// TwinCAT 3 PLC project Lynus_Test
// ProgramVersion: 3.1.4023.0
// libraries:
//   EfficientIO Communicator, * (EfficientIO)
//   EfficientIO ModbusTCP, * (EfficientIO)
//   Lynus Standards, * (Lynus AG)
//   Tc2_ModbusSrv, * (Beckhoff Automation GmbH)
//   Tc2_Standard, * (Beckhoff Automation GmbH)
//   Tc2_System, * (Beckhoff Automation GmbH)
//   Tc2_Utilities, * (Beckhoff Automation GmbH)
//   Tc3_Module, * (Beckhoff Automation GmbH)
//   Lynus Energy Basic,1.0.0.2,Lynus AG
// project tree:
//   DUTs/ st_P_Connect_to_Lynus.TcDUT
//   GVLs/ GVL.TcGVL, p_Datenschnittstelle_L.TcPOU
//   Lynus/ EfficientIO_Read_Wirte.TcPOU, MqttCommunicator.TcPOU, PrgEMS.TcPOU, PrgModbus.TcPOU, p_call_fast_task.TcPOU, p_slow_task.TcPOU
//   / EfficientIO_Communication.TcTTO, PlcTask1.TcTTO
// (motion and I/O tree: see PLC project p_connect)
// real-time tasks:
//   TASK PlcTask: cycle T#10ms, priority 20, ADS port 350
//   TASK EfficientIO_Communication: cycle T#5ms, priority 15, ADS port 351
//   TASK PlcTask1: cycle T#10ms, priority 21, ADS port 353
// variable links:
//   Lynus_Test/Lynus_Test Instance <-> P_Connect/P_Connect Instance
//     PlcTask1 Inputs/GVL.lynus_in <-> PlcTask Outputs/GVL_EfficientIO.lynus_out
//     PlcTask1 Outputs/GVL.lynus_out <-> PlcTask Inputs/GVL_EfficientIO.lynus_in

CONFIGURATION Lynus_Test
    RESOURCE PLC ON TwinCAT3
        TASK EfficientIO_Communication(INTERVAL := T#5ms, PRIORITY := 15);
        TASK PlcTask1(INTERVAL := T#10ms, PRIORITY := 21);
        PROGRAM p_call_fast_task WITH EfficientIO_Communication : p_call_fast_task;
        PROGRAM p_slow_task WITH PlcTask1 : p_slow_task;
    END_RESOURCE
END_CONFIGURATION

// ---- DUTs/st_P_Connect_to_Lynus.TcDUT
TYPE st_P_Connect_to_Lynus :
STRUCT
	Wert_1	:REAL;	
	Wert_2	:REAL;	
	Wert_3	:REAL;	
	Wert_4	:REAL;	
	Wert_5	:REAL;	
	Wert_6	:REAL;	
	Wert_7	:BOOL;	
	Wert_8	:REAL;	
	Wert_9	:REAL;	
	Wert_10	:REAL;
	Wert_11	:REAL;	
	Wert_12	:REAL;	
	Wert_13	:REAL;	
	Wert_14	:REAL;	
	Wert_15	:REAL;	
	Wert_16	:REAL;	
	Wert_17	:REAL;	
	Wert_18	:REAL;	
	Wert_19	:REAL;	
	Wert_20	:REAL;
	Wert_21	:REAL;	
	Wert_22	:REAL;	
	Wert_23	:REAL;	
	Wert_24	:REAL;	
	Wert_25	:REAL;	
	Wert_26	:REAL;	
	Wert_27	:REAL;	
	Wert_28	:REAL;	
	Wert_29	:REAL;	
	Wert_30	:REAL;
	Wert_31	:REAL;
	Wert_32	:REAL;
	Wert_33	:REAL;
	Wert_34	:REAL;
	Wert_35	:REAL;
	Wert_36	:REAL;
	Wert_37	:REAL;
	Wert_38	:REAL;
	Wert_39	:REAL;
	Wert_40	:REAL;
	Wert_41	:BOOL;
	Wert_42	:BOOL;
	Wert_43	:BOOL;
	Wert_44	:BOOL;
	Wert_45	:BOOL;
	Wert_46	:BOOL;
	Wert_47	:BOOL;
	Wert_48	:BOOL;
	Wert_49	:BOOL;
	Wert_50	:BOOL;
	Wert_51	:BOOL;
	Wert_52	:BOOL;
END_STRUCT
END_TYPE

// ---- GVLs/GVL.TcGVL
{attribute 'qualified_only'}
VAR_GLOBAL
	lynus_in   				AT %I* 	: st_P_Connect_to_Lynus;
	lynus_out   			AT %Q* 	: st_P_Connect_to_Lynus;
	
	NULL						:REAL;//{#lynus.ag#()}
	
	(*KNX*)
	TEMP_INNEN_1					:REAL;//{#lynus.ag#()}
	RH_INNEN_1						:REAL;//{#lynus.ag#()}
	TEMP_INNEN_2					:REAL;//{#lynus.ag#()}
	RH_INNEN_2						:REAL;//{#lynus.ag#()}
	TEMP_AUSSEN						:REAL;//{#lynus.ag#()}
	RH_AUSSEN						:REAL;//{#lynus.ag#()}
	AKTIVITAET						:BOOL;//{#lynus.ag#()}
	
	(*M-Bus variablen für Lynus*)
	ELEKTRO_1_Zaehler		:REAL;//{#lynus.ag#()}
	ELEKTRO_1_Leistung		:REAL;//{#lynus.ag#()}
	ELEKTRO_2_Zaehler		:REAL;//{#lynus.ag#()}
	ELEKTRO_2_Leistung		:REAL;//{#lynus.ag#()}
	ELEKTRO_3_Zaehler		:REAL;//{#lynus.ag#()}
	ELEKTRO_3_Leistung		:REAL;//{#lynus.ag#()}
	ELEKTRO_4_Zaehler		:REAL;//{#lynus.ag#()}
	ELEKTRO_4_Leistung		:REAL;//{#lynus.ag#()}
	ELEKTRO_5_Zaehler		:REAL;//{#lynus.ag#()}
	ELEKTRO_5_Leistung		:REAL;//{#lynus.ag#()}
	HEIZEN					:REAL;//{#lynus.ag#()}
	HEIZEN_E_Lesitung		:REAL;//{#lynus.ag#()}
	
	(*IMPULSZÄHLER*)
	Wasseruhr_1				:REAL;//{#lynus.ag#()}
	Wasseruhr_2				:REAL;//{#lynus.ag#()}

	(*PT1000 Temp.*)
	TEMP_HKLS_1				:REAL;//{#lynus.ag#()}
	TEMP_HKLS_2				:REAL;//{#lynus.ag#()}
	TEMP_HKLS_3				:REAL;//{#lynus.ag#()}
	TEMP_HKLS_4				:REAL;//{#lynus.ag#()}
	TEMP_HKLS_5				:REAL;//{#lynus.ag#()}
	TEMP_HKLS_6				:REAL;//{#lynus.ag#()}
	TEMP_HKLS_7				:REAL;//{#lynus.ag#()}
	TEMP_HKLS_8				:REAL;//{#lynus.ag#()}
	
	(*Zentalfunktionen*)
	VERSCHATTUNG_auf		:BOOL;//{#lynus.ag#()}
	VERSCHATTUNG_ab			:BOOL;//{#lynus.ag#()}
	ZENTRAL_LICHT_ein_EG	:BOOL;//{#lynus.ag#()}
	ZENTRAL_LICHT_aus_EG	:BOOL;//{#lynus.ag#()}
	ZENTRAL_LICHT_ein_OG	:BOOL;//{#lynus.ag#()}
	ZENTRAL_LICHT_aus_OG	:BOOL;//{#lynus.ag#()}
	B3_ZENTRAL_LICHT_ein	:BOOL;//{#lynus.ag#()}
	B3_ZENTRAL_LICHT_aus	:BOOL;//{#lynus.ag#()}
	B3_SCHATTUNG_auf_EG		:BOOL;//{#lynus.ag#()}
	B3_SCHATTUNG_ab_EG		:BOOL;//{#lynus.ag#()}
	B3_SCHATTUNG_auf_OG		:BOOL;//{#lynus.ag#()}
	B3_SCHATTUNG_ab_OG		:BOOL;//{#lynus.ag#()}
	
	Wert_30					:REAL;//{#lynus.ag#()}
	Wert_31					:REAL;//{#lynus.ag#()}
	Wert_32					:REAL;//{#lynus.ag#()}
	Wert_33					:REAL;//{#lynus.ag#()}
	dummy_					:BOOL;//{#lynus.ag#()}
END_VAR

// ---- Lynus/p_call_fast_task.TcPOU
PROGRAM p_call_fast_task
VAR
	EfficientIO: INT;
END_VAR

(* Es wird standartmäßig M-Bus verwendet, bei IMMODO wurden Mod-Bus zähler verbaut *)
//Communication_KL6781();
(*MAIN_Zaehlerbaustein()*);

(*FB's von Lynus die den FastTask bennötigen*)
EfficientIO_Read_Wirte();

END_PROGRAM

// ---- Lynus/EfficientIO_Read_Wirte.TcPOU
PROGRAM EfficientIO_Read_Wirte
VAR
	fbVar				: FB_VarInfo;
	fbRW				: FB_ReadWrite;
END_VAR

(*Der FB_VarInfo sammelt die Informationen über alle kommentierten Variablen in der SPS.*)
fbVar(
	bReadInfo:= , 
	eTMCFile:= eSelectTMCFile.eDontUseTMCFile, 
	eSavePositionTMCFile:= eSavePositionOnPLC.ePostionC, 
	udiCounterFoundVariables=> , 
	bError=> , 
	bBusy=> , 
	byProgress=> , 
	udiErrorCodeOut=> , 
	eErrorVarInfo_Out=> , 
	sVarWithError=> );

(*Der FB_ReadWrite dient nach dem Scannen der Symbole dem Lesen und Schreiben der Werte.
Die gelesenen Werte werden in Richtung Cloud geschickt und die schreibenden, kommend von
der Cloud, werden auf den Wert der SPS geschrieben.*)
fbrw();

END_PROGRAM

// ---- Lynus/p_slow_task.TcPOU
PROGRAM p_slow_task
VAR
END_VAR

(*Programmaufrufte im slow Task (10ms)*)
//Call Slow Tasks for Lynus 	
MqttCommunicator();
p_Datenschnittstelle_L();


//Stefan Lackner 14.02.2023
PrgModbus();		// Modbus TCP functions
PrgEMS();			// EMS Fucntion

END_PROGRAM

// ---- Lynus/MqttCommunicator.TcPOU
PROGRAM MqttCommunicator
VAR
	fbCom			: FB_MqttCommunicator_V5;
END_VAR

(*notdonepoint Bitte UserName und UserPassword eintragen, dies bekommt man direkt von der LynusWebsite*)
fbCom(
	bConnect:= TRUE, 
	strAuthKey:= 'ENE87365342998', 
	sUserName:='7ad7b8b6-0630-4d31-a3b5-e626a3dca2b4', 
	sUserPassword:='b0a3873e-12bb-4efd-a1d1-df77771e0e45', 
	eSavePositionCertificate:= eSavePositionOnPLC.ePostionC, 
	bConnected=> , 
	bError=> , 
	hrErrorCode=> , 
	eConnectionState=> , 
	eErrorMessage_Out=> );

(*fbCom(
	bConnect:= TRUE, 
	sUserName:= '0d553fc2-e7f3-4571-9008-fb5428f4c828',
	sUserPassword:= '8604f195-2f00-444b-ac81-e02a496b91e8', 
	eSavePositionCertificate:= eSavePositionOnPLC.ePostionC, 
	bConnected=> , 
	bError=> , 
	hrErrorCode=> , 
	eConnectionState=> , 
	eErrorMessage_Out=> );
	*)

END_PROGRAM

// ---- GVLs/p_Datenschnittstelle_L.TcPOU
PROGRAM p_Datenschnittstelle_L
VAR
END_VAR

GVL.NULL				:=0.0;
GVL.TEMP_INNEN_1		:= GVL.lynus_in.Wert_1;	
GVL.RH_INNEN_1			:= GVL.lynus_in.Wert_2;
GVL.TEMP_INNEN_2		:= GVL.lynus_in.Wert_3;
GVL.RH_INNEN_2			:= GVL.lynus_in.Wert_4;
GVL.TEMP_AUSSEN			:= GVL.lynus_in.Wert_5;
GVL.RH_AUSSEN			:= GVL.lynus_in.Wert_6;
GVL.AKTIVITAET			:= GVL.lynus_in.Wert_7;
GVL.ELEKTRO_1_Zaehler	:= GVL.lynus_in.Wert_8;
GVL.ELEKTRO_1_Leistung	:= GVL.lynus_in.Wert_9;
GVL.ELEKTRO_2_Zaehler	:= GVL.lynus_in.Wert_10;
GVL.ELEKTRO_2_Leistung	:= GVL.lynus_in.Wert_11;
GVL.ELEKTRO_3_Zaehler	:= GVL.lynus_in.Wert_12;
GVL.ELEKTRO_3_Leistung	:= GVL.lynus_in.Wert_13;
GVL.ELEKTRO_4_Zaehler	:= GVL.lynus_in.Wert_14;
GVL.ELEKTRO_4_Leistung	:= GVL.lynus_in.Wert_15;
GVL.ELEKTRO_5_Zaehler	:= GVL.lynus_in.Wert_16;
GVL.ELEKTRO_5_Leistung	:= GVL.lynus_in.Wert_17;
GVL.HEIZEN				:= GVL.lynus_in.Wert_18;
GVL.HEIZEN_E_Lesitung	:= GVL.lynus_in.Wert_19;
GVL.Wasseruhr_1			:= GVL.lynus_in.Wert_20;
GVL.Wasseruhr_2			:= GVL.lynus_in.Wert_21;
GVL.TEMP_HKLS_1			:= GVL.lynus_in.Wert_22;
GVL.TEMP_HKLS_2			:= GVL.lynus_in.Wert_23;
GVL.TEMP_HKLS_3			:= GVL.lynus_in.Wert_24;
GVL.TEMP_HKLS_4			:= GVL.lynus_in.Wert_25;
GVL.TEMP_HKLS_5			:= GVL.lynus_in.Wert_26;
GVL.TEMP_HKLS_6			:= GVL.lynus_in.Wert_27;
GVL.TEMP_HKLS_7			:= GVL.lynus_in.Wert_28;
GVL.TEMP_HKLS_8			:= GVL.lynus_in.Wert_29;

GVL.Wert_30				:= GVL.lynus_in.Wert_30;
GVL.Wert_31				:= GVL.lynus_in.Wert_31; //BA3 WP Leistung
GVL.Wert_32				:= GVL.lynus_in.Wert_32; //BA3 WP Energie Wärme
GVL.Wert_33				:= GVL.lynus_in.Wert_33; //BA3 WP Energie Kälte

GVL.lynus_out.Wert_41	:= GVL.VERSCHATTUNG_auf;
GVL.lynus_out.Wert_42	:= GVL.VERSCHATTUNG_ab;
GVL.lynus_out.Wert_43	:= GVL.ZENTRAL_LICHT_ein_EG;
GVL.lynus_out.Wert_44	:= GVL.ZENTRAL_LICHT_aus_EG;
GVL.lynus_out.Wert_45	:= GVL.ZENTRAL_LICHT_ein_OG;
GVL.lynus_out.Wert_46	:= GVL.ZENTRAL_LICHT_aus_OG;
GVL.lynus_out.Wert_47	:= GVL.B3_ZENTRAL_LICHT_ein;
GVL.lynus_out.Wert_48	:= GVL.B3_ZENTRAL_LICHT_aus;
GVL.lynus_out.Wert_49	:= GVL.B3_SCHATTUNG_auf_EG;
GVL.lynus_out.Wert_50	:= GVL.B3_SCHATTUNG_ab_EG;
GVL.lynus_out.Wert_51	:= GVL.B3_SCHATTUNG_auf_OG;
GVL.lynus_out.Wert_52	:= GVL.B3_SCHATTUNG_ab_OG;

END_PROGRAM

// ---- Lynus/PrgModbus.TcPOU
PROGRAM PrgModbus
VAR
	FB_KEBA_CS1				:FB_ECS_KEBA_P30;
	FB_Schneider_EVLink_1	:FB_Schneider_EVlinkWallbox;
	FB_Schneider_EVLink_2	:FB_Schneider_EVlinkWallbox;
	FB_Schneider_EVLink_3	:FB_Schneider_EVlinkWallbox;
	FB_Schneider_EVLink_4	:FB_Schneider_EVlinkWallbox;
	FB_Schneider_EVLink_5	:FB_Schneider_EVlinkWallbox;
	FB_Schneider_EVLink_6	:FB_Schneider_EVlinkWallbox;
	FB_Schneider_EVLink_7	:FB_Schneider_EVlinkWallbox;
	FB_Schneider_EVLink_8	:FB_Schneider_EVlinkWallbox;
	FB_Schneider_EVLink_9	:FB_Schneider_EVlinkWallbox;
	FB_Schneider_EVLink_10	:FB_Schneider_EVlinkWallbox;
	FB_Schneider_EVLink_11	:FB_Schneider_EVlinkWallbox;
	FB_Schneider_EVLink_12	:FB_Schneider_EVlinkWallbox;
	FB_Schneider_EVLink_13	:FB_Schneider_EVlinkWallbox;
	FB_Schneider_EVLink_14	:FB_Schneider_EVlinkWallbox;
	FB_Schneider_EVLink_15	:FB_Schneider_EVlinkWallbox;
	FB_Schneider_EVLink_16	:FB_Schneider_EVlinkWallbox;
	FB_Schneider_EVLink_17	:FB_Schneider_EVlinkWallbox;
	FB_Schneider_EVLink_18	:FB_Schneider_EVlinkWallbox;
	lr_CSPowerTotal: LREAL;													//{#lynus.ag#()}
	lr_CSPower_1: LREAL;													//{#lynus.ag#()}
	lr_CSPower_2: LREAL;													//{#lynus.ag#()}
	lr_CSPower_3: LREAL;													//{#lynus.ag#()}
	lr_CSPower_4: LREAL;													//{#lynus.ag#()}
	lr_CSPower_5: LREAL;													//{#lynus.ag#()}
	lr_CSPower_6: LREAL;													//{#lynus.ag#()}
	lr_CSPower_7: LREAL;													//{#lynus.ag#()}
	lr_CSPower_8: LREAL;													//{#lynus.ag#()}
	lr_CSPower_9: LREAL;													//{#lynus.ag#()}
	lr_CSPower_10: LREAL;													//{#lynus.ag#()}
	lr_CSPower_11: LREAL;													//{#lynus.ag#()}
	lr_CSPower_12: LREAL;													//{#lynus.ag#()}
	lr_CSPower_13: LREAL;													//{#lynus.ag#()}
	lr_CSPower_14: LREAL;													//{#lynus.ag#()}
	lr_CSPower_15: LREAL;													//{#lynus.ag#()}
	lr_CSPower_16: LREAL;													//{#lynus.ag#()}
	lr_CSPower_17: LREAL;													//{#lynus.ag#()}
	lr_CSPower_18: LREAL;													//{#lynus.ag#()}
 	lr_CSEnergy_Total: LREAL;												//{#lynus.ag#()}
	bIsEnabledCS_1			: BOOL;									//{#lynus.ag#()}
	byErrorWarningCS_1		: BYTE;									//{#lynus.ag#()}
	byStateMinPowerCS_1		: BYTE;									//{#lynus.ag#()}
	rTargetPowerCS_1		: REAL;									//{#lynus.ag#()}
	bCarConnectedCS_1		: BOOL;									//{#lynus.ag#()}
	rChrgTimeCS_1			: REAL;									//{#lynus.ag#()}
	byChrgManuSPCS_1		: BYTE;									//{#lynus.ag#()}
	bChrgManuCS_1			: bool;									//{#lynus.ag#()}
	bStateOkCS_1			: BOOL;									//{#lynus.ag#()}
	bIsEnabledCS_2			: BOOL;									//{#lynus.ag#()}
	byErrorWarningCS_2		: BYTE;									//{#lynus.ag#()}
	byStateMinPowerCS_2		: BYTE;									//{#lynus.ag#()}
	rTargetPowerCS_2		: REAL;									//{#lynus.ag#()}
	bCarConnectedCS_2		: BOOL;									//{#lynus.ag#()}
	rChrgTimeCS_2			: REAL;									//{#lynus.ag#()}
	byChrgManuSPCS_2		: BYTE;									//{#lynus.ag#()}
	bChrgManuCS_2			: bool;									//{#lynus.ag#()}
	bStateOkCS_2			: BOOL;									//{#lynus.ag#()}
	bIsEnabledCS_3			: BOOL;									//{#lynus.ag#()}
	byErrorWarningCS_3		: BYTE;									//{#lynus.ag#()}
	byStateMinPowerCS_3		: BYTE;									//{#lynus.ag#()}
	rTargetPowerCS_3		: REAL;									//{#lynus.ag#()}
	bCarConnectedCS_3		: BOOL;									//{#lynus.ag#()}
	rChrgTimeCS_3			: REAL;									//{#lynus.ag#()}
	byChrgManuSPCS_3		: BYTE;									//{#lynus.ag#()}
	bChrgManuCS_3			: BOOL;									//{#lynus.ag#()}
	bStateOkCS_3			: BOOL;									//{#lynus.ag#()}
	bIsEnabledCS_4			: BOOL;									//{#lynus.ag#()}
	byErrorWarningCS_4		: BYTE;									//{#lynus.ag#()}
	byStateMinPowerCS_4		: BYTE;									//{#lynus.ag#()}
	rTargetPowerCS_4		: REAL;									//{#lynus.ag#()}
	bCarConnectedCS_4		: BOOL;									//{#lynus.ag#()}
	rChrgTimeCS_4			: REAL;									//{#lynus.ag#()}
	byChrgManuSPCS_4		: BYTE;									//{#lynus.ag#()}
	bChrgManuCS_4			: BOOL;									//{#lynus.ag#()}
	bStateOkCS_4			: BOOL;									//{#lynus.ag#()}
	bIsEnabledCS_5			: BOOL;									//{#lynus.ag#()}
	byErrorWarningCS_5		: BYTE;									//{#lynus.ag#()}
	byStateMinPowerCS_5		: BYTE;									//{#lynus.ag#()}
	rTargetPowerCS_5		: REAL;									//{#lynus.ag#()}
	bCarConnectedCS_5		: BOOL;									//{#lynus.ag#()}
	rChrgTimeCS_5			: REAL;									//{#lynus.ag#()}
	byChrgManuSPCS_5		: BYTE;									//{#lynus.ag#()}
	bChrgManuCS_5			: BOOL;									//{#lynus.ag#()}
	bStateOkCS_5			: BOOL;									//{#lynus.ag#()}
	bIsEnabledCS_6			: BOOL;									//{#lynus.ag#()}
	byErrorWarningCS_6		: BYTE;									//{#lynus.ag#()}
	byStateMinPowerCS_6		: BYTE;									//{#lynus.ag#()}
	rTargetPowerCS_6		: REAL;									//{#lynus.ag#()}
	bCarConnectedCS_6		: BOOL;									//{#lynus.ag#()}
	rChrgTimeCS_6			: REAL;									//{#lynus.ag#()}
	byChrgManuSPCS_6		: BYTE;									//{#lynus.ag#()}
	bChrgManuCS_6			: BOOL;									//{#lynus.ag#()}
	bStateOkCS_6			: BOOL;									//{#lynus.ag#()}
	bIsEnabledCS_7			: BOOL;									//{#lynus.ag#()}
	byErrorWarningCS_7		: BYTE;									//{#lynus.ag#()}
	byStateMinPowerCS_7		: BYTE;									//{#lynus.ag#()}
	rTargetPowerCS_7		: REAL;									//{#lynus.ag#()}
	bCarConnectedCS_7		: BOOL;									//{#lynus.ag#()}
	rChrgTimeCS_7			: REAL;									//{#lynus.ag#()}
	byChrgManuSPCS_7		: BYTE;									//{#lynus.ag#()}
	bChrgManuCS_7			: BOOL;									//{#lynus.ag#()}
	bStateOkCS_7			: BOOL;									//{#lynus.ag#()}
	bIsEnabledCS_8			: BOOL;									//{#lynus.ag#()}
	byErrorWarningCS_8		: BYTE;									//{#lynus.ag#()}
	byStateMinPowerCS_8		: BYTE;									//{#lynus.ag#()}
	rTargetPowerCS_8		: REAL;									//{#lynus.ag#()}
	bCarConnectedCS_8		: BOOL;									//{#lynus.ag#()}
	rChrgTimeCS_8			: REAL;									//{#lynus.ag#()}
	byChrgManuSPCS_8		: BYTE;									//{#lynus.ag#()}
	bChrgManuCS_8			: BOOL;									//{#lynus.ag#()}
	bStateOkCS_8			: BOOL;									//{#lynus.ag#()}
	bIsEnabledCS_9			: BOOL;									//{#lynus.ag#()}
	byErrorWarningCS_9		: BYTE;									//{#lynus.ag#()}
	byStateMinPowerCS_9		: BYTE;									//{#lynus.ag#()}
	rTargetPowerCS_9		: REAL;									//{#lynus.ag#()}
	bCarConnectedCS_9		: BOOL;									//{#lynus.ag#()}
	rChrgTimeCS_9			: REAL;									//{#lynus.ag#()}
	byChrgManuSPCS_9		: BYTE;									//{#lynus.ag#()}
	bChrgManuCS_9			: BOOL;									//{#lynus.ag#()}
	bStateOkCS_9			: BOOL;									//{#lynus.ag#()}
	bIsEnabledCS_10			: BOOL;									//{#lynus.ag#()}
	byErrorWarningCS_10		: BYTE;									//{#lynus.ag#()}
	byStateMinPowerCS_10	: BYTE;									//{#lynus.ag#()}
	rTargetPowerCS_10		: REAL;									//{#lynus.ag#()}
	bCarConnectedCS_10		: BOOL;									//{#lynus.ag#()}
	rChrgTimeCS_10			: REAL;									//{#lynus.ag#()}
	byChrgManuSPCS_10		: BYTE;									//{#lynus.ag#()}
	bChrgManuCS_10			: BOOL;									//{#lynus.ag#()}
	bStateOkCS_10			: BOOL;									//{#lynus.ag#()}
	bIsEnabledCS_11			: BOOL;									//{#lynus.ag#()}
	byErrorWarningCS_11		: BYTE;									//{#lynus.ag#()}
	byStateMinPowerCS_11	: BYTE;									//{#lynus.ag#()}
	rTargetPowerCS_11		: REAL;									//{#lynus.ag#()}
	bCarConnectedCS_11		: BOOL;									//{#lynus.ag#()}
	rChrgTimeCS_11			: REAL;									//{#lynus.ag#()}
	byChrgManuSPCS_11		: BYTE;									//{#lynus.ag#()}
	bChrgManuCS_11			: BOOL;									//{#lynus.ag#()}
	bStateOkCS_11			: BOOL;									//{#lynus.ag#()}
	bIsEnabledCS_12			: BOOL;									//{#lynus.ag#()}
	byErrorWarningCS_12		: BYTE;									//{#lynus.ag#()}
	byStateMinPowerCS_12	: BYTE;									//{#lynus.ag#()}
	rTargetPowerCS_12		: REAL;									//{#lynus.ag#()}
	bCarConnectedCS_12		: BOOL;									//{#lynus.ag#()}
	rChrgTimeCS_12			: REAL;									//{#lynus.ag#()}
	byChrgManuSPCS_12		: BYTE;									//{#lynus.ag#()}
	bChrgManuCS_12			: BOOL;									//{#lynus.ag#()}
	bStateOkCS_12			: BOOL;									//{#lynus.ag#()}
	bIsEnabledCS_13			: BOOL;									//{#lynus.ag#()}
	byErrorWarningCS_13		: BYTE;									//{#lynus.ag#()}
	byStateMinPowerCS_13	: BYTE;									//{#lynus.ag#()}
	rTargetPowerCS_13		: REAL;									//{#lynus.ag#()}
	bCarConnectedCS_13		: BOOL;									//{#lynus.ag#()}
	rChrgTimeCS_13			: REAL;									//{#lynus.ag#()}
	byChrgManuSPCS_13		: BYTE;									//{#lynus.ag#()}
	bChrgManuCS_13			: BOOL;									//{#lynus.ag#()}
	bStateOkCS_13			: BOOL;									//{#lynus.ag#()}
	bIsEnabledCS_14			: BOOL;									//{#lynus.ag#()}
	byErrorWarningCS_14		: BYTE;									//{#lynus.ag#()}
	byStateMinPowerCS_14	: BYTE;									//{#lynus.ag#()}
	rTargetPowerCS_14		: REAL;									//{#lynus.ag#()}
	bCarConnectedCS_14		: BOOL;									//{#lynus.ag#()}
	rChrgTimeCS_14			: REAL;									//{#lynus.ag#()}
	byChrgManuSPCS_14		: BYTE;									//{#lynus.ag#()}
	bChrgManuCS_14			: BOOL;									//{#lynus.ag#()}
	bStateOkCS_14			: BOOL;									//{#lynus.ag#()}
	bIsEnabledCS_15			: BOOL;									//{#lynus.ag#()}
	byErrorWarningCS_15		: BYTE;									//{#lynus.ag#()}
	byStateMinPowerCS_15	: BYTE;									//{#lynus.ag#()}
	rTargetPowerCS_15		: REAL;									//{#lynus.ag#()}
	bCarConnectedCS_15		: BOOL;									//{#lynus.ag#()}
	rChrgTimeCS_15			: REAL;									//{#lynus.ag#()}
	byChrgManuSPCS_15		: BYTE;									//{#lynus.ag#()}
	bChrgManuCS_15			: BOOL;									//{#lynus.ag#()}
	bStateOkCS_15			: BOOL;									//{#lynus.ag#()}
	bIsEnabledCS_16			: BOOL;									//{#lynus.ag#()}
	byErrorWarningCS_16		: BYTE;									//{#lynus.ag#()}
	byStateMinPowerCS_16	: BYTE;									//{#lynus.ag#()}
	rTargetPowerCS_16		: REAL;									//{#lynus.ag#()}
	bCarConnectedCS_16		: BOOL;									//{#lynus.ag#()}
	rChrgTimeCS_16			: REAL;									//{#lynus.ag#()}
	byChrgManuSPCS_16		: BYTE;									//{#lynus.ag#()}
	bChrgManuCS_16			: BOOL;									//{#lynus.ag#()}
	bStateOkCS_16			: BOOL;									//{#lynus.ag#()}
	bIsEnabledCS_17			: BOOL;									//{#lynus.ag#()}
	byErrorWarningCS_17		: BYTE;									//{#lynus.ag#()}
	byStateMinPowerCS_17	: BYTE;									//{#lynus.ag#()}
	rTargetPowerCS_17		: REAL;									//{#lynus.ag#()}
	bCarConnectedCS_17		: BOOL;									//{#lynus.ag#()}
	rChrgTimeCS_17			: REAL;									//{#lynus.ag#()}
	byChrgManuSPCS_17		: BYTE;									//{#lynus.ag#()}
	bChrgManuCS_17			: BOOL;									//{#lynus.ag#()}
	bStateOkCS_17			: BOOL;									//{#lynus.ag#()}
	bIsEnabledCS_18			: BOOL;									//{#lynus.ag#()}
	byErrorWarningCS_18		: BYTE;									//{#lynus.ag#()}
	byStateMinPowerCS_18	: BYTE;									//{#lynus.ag#()}
	rTargetPowerCS_18		: REAL;									//{#lynus.ag#()}
	bCarConnectedCS_18		: BOOL;									//{#lynus.ag#()}
	rChrgTimeCS_18			: REAL;									//{#lynus.ag#()}
	byChrgManuSPCS_18		: BYTE;									//{#lynus.ag#()}
	bChrgManuCS_18			: BOOL;									//{#lynus.ag#()}
	bStateOkCS_18			: BOOL;									//{#lynus.ag#()}
	r_House: REAL;													//{#lynus.ag#()}
	lr_EnergyCounterCS_1	: REAL;									//{#lynus.ag#()}
	lr_EnergyCounterCS_2	: REAL;									//{#lynus.ag#()}
	lr_EnergyCounterCS_3	: REAL;									//{#lynus.ag#()}
	lr_EnergyCounterCS_4	: REAL;									//{#lynus.ag#()}
	lr_EnergyCounterCS_5	: REAL;									//{#lynus.ag#()}
	lr_EnergyCounterCS_6	: REAL;									//{#lynus.ag#()}
	lr_EnergyCounterCS_7	: REAL;									//{#lynus.ag#()}
	lr_EnergyCounterCS_8	: REAL;									//{#lynus.ag#()}
	lr_EnergyCounterCS_9	: REAL;									//{#lynus.ag#()}
	lr_EnergyCounterCS_10	: REAL;									//{#lynus.ag#()}
	lr_EnergyCounterCS_11	: REAL;									//{#lynus.ag#()}
	lr_EnergyCounterCS_12	: REAL;									//{#lynus.ag#()}
	lr_EnergyCounterCS_13	: REAL;									//{#lynus.ag#()}
	lr_EnergyCounterCS_14	: REAL;									//{#lynus.ag#()}
	lr_EnergyCounterCS_15	: REAL;									//{#lynus.ag#()}
	lr_EnergyCounterCS_16	: REAL;									//{#lynus.ag#()}
	lr_EnergyCounterCS_17	: REAL;									//{#lynus.ag#()}
	lr_EnergyCounterCS_18	: REAL;									//{#lynus.ag#()}


END_VAR
VAR PERSISTENT
	bEnabledCS_1			: BOOL;									//{#lynus.ag#()}
	byPrioCS_1				: BYTE;									//{#lynus.ag#()}
	bySOC_E_CS_1			: BYTE;									//{#lynus.ag#()}
	bySOC_D_CS_1			: BYTE;									//{#lynus.ag#()}
	byMinPowerCS_1			: BYTE;									//{#lynus.ag#()}
	rMaxPowerCS_1			: REAL;									//{#lynus.ag#()}
	bEnabledCS_2			: BOOL;									//{#lynus.ag#()}
	byPrioCS_2				: BYTE;									//{#lynus.ag#()}
	bySOC_E_CS_2			: BYTE;									//{#lynus.ag#()}
	bySOC_D_CS_2			: BYTE;									//{#lynus.ag#()}
	byMinPowerCS_2			: BYTE;									//{#lynus.ag#()}
	rMaxPowerCS_2			: REAL;									//{#lynus.ag#()}
	bEnabledCS_3			: BOOL;									//{#lynus.ag#()}
	byPrioCS_3				: BYTE;									//{#lynus.ag#()}
	bySOC_E_CS_3			: BYTE;									//{#lynus.ag#()}
	bySOC_D_CS_3			: BYTE;									//{#lynus.ag#()}
	byMinPowerCS_3			: BYTE;									//{#lynus.ag#()}
	rMaxPowerCS_3			: REAL;									//{#lynus.ag#()}
	bEnabledCS_4			: BOOL;									//{#lynus.ag#()}
	byPrioCS_4				: BYTE;									//{#lynus.ag#()}
	bySOC_E_CS_4			: BYTE;									//{#lynus.ag#()}
	bySOC_D_CS_4			: BYTE;									//{#lynus.ag#()}
	byMinPowerCS_4			: BYTE;									//{#lynus.ag#()}
	rMaxPowerCS_4			: REAL;									//{#lynus.ag#()}
	bEnabledCS_5			: BOOL;									//{#lynus.ag#()}
	byPrioCS_5				: BYTE;									//{#lynus.ag#()}
	bySOC_E_CS_5			: BYTE;									//{#lynus.ag#()}
	bySOC_D_CS_5			: BYTE;									//{#lynus.ag#()}
	byMinPowerCS_5			: BYTE;									//{#lynus.ag#()}
	rMaxPowerCS_5			: REAL;									//{#lynus.ag#()}
	bEnabledCS_6			: BOOL;									//{#lynus.ag#()}
	byPrioCS_6				: BYTE;									//{#lynus.ag#()}
	bySOC_E_CS_6			: BYTE;									//{#lynus.ag#()}
	bySOC_D_CS_6			: BYTE;									//{#lynus.ag#()}
	byMinPowerCS_6			: BYTE;									//{#lynus.ag#()}
	rMaxPowerCS_6			: REAL;									//{#lynus.ag#()}
	bEnabledCS_7			: BOOL;									//{#lynus.ag#()}
	byPrioCS_7				: BYTE;									//{#lynus.ag#()}
	bySOC_E_CS_7			: BYTE;									//{#lynus.ag#()}
	bySOC_D_CS_7			: BYTE;									//{#lynus.ag#()}
	byMinPowerCS_7			: BYTE;									//{#lynus.ag#()}
	rMaxPowerCS_7			: REAL;									//{#lynus.ag#()}
	bEnabledCS_8			: BOOL;									//{#lynus.ag#()}
	byPrioCS_8				: BYTE;									//{#lynus.ag#()}
	bySOC_E_CS_8			: BYTE;									//{#lynus.ag#()}
	bySOC_D_CS_8			: BYTE;									//{#lynus.ag#()}
	byMinPowerCS_8			: BYTE;									//{#lynus.ag#()}
	rMaxPowerCS_8			: REAL;									//{#lynus.ag#()}
	bEnabledCS_9			: BOOL;									//{#lynus.ag#()}
	byPrioCS_9				: BYTE;									//{#lynus.ag#()}
	bySOC_E_CS_9			: BYTE;									//{#lynus.ag#()}
	bySOC_D_CS_9			: BYTE;									//{#lynus.ag#()}
	byMinPowerCS_9			: BYTE;									//{#lynus.ag#()}
	rMaxPowerCS_9			: REAL;									//{#lynus.ag#()}
	bEnabledCS_10			: BOOL;									//{#lynus.ag#()}
	byPrioCS_10				: BYTE;									//{#lynus.ag#()}
	bySOC_E_CS_10			: BYTE;									//{#lynus.ag#()}
	bySOC_D_CS_10			: BYTE;									//{#lynus.ag#()}
	byMinPowerCS_10			: BYTE;									//{#lynus.ag#()}
	rMaxPowerCS_10			: REAL;									//{#lynus.ag#()}
	bEnabledCS_11			: BOOL;									//{#lynus.ag#()}
	byPrioCS_11				: BYTE;									//{#lynus.ag#()}
	bySOC_E_CS_11			: BYTE;									//{#lynus.ag#()}
	bySOC_D_CS_11			: BYTE;									//{#lynus.ag#()}
	byMinPowerCS_11			: BYTE;									//{#lynus.ag#()}
	rMaxPowerCS_11			: REAL;									//{#lynus.ag#()}
	bEnabledCS_12			: BOOL;									//{#lynus.ag#()}
	byPrioCS_12				: BYTE;									//{#lynus.ag#()}
	bySOC_E_CS_12			: BYTE;									//{#lynus.ag#()}
	bySOC_D_CS_12			: BYTE;									//{#lynus.ag#()}
	byMinPowerCS_12			: BYTE;									//{#lynus.ag#()}
	rMaxPowerCS_12			: REAL;									//{#lynus.ag#()}
	bEnabledCS_13			: BOOL;									//{#lynus.ag#()}
	byPrioCS_13				: BYTE;									//{#lynus.ag#()}
	bySOC_E_CS_13			: BYTE;									//{#lynus.ag#()}
	bySOC_D_CS_13			: BYTE;									//{#lynus.ag#()}
	byMinPowerCS_13			: BYTE;									//{#lynus.ag#()}
	rMaxPowerCS_13			: REAL;									//{#lynus.ag#()}
	bEnabledCS_14			: BOOL;									//{#lynus.ag#()}
	byPrioCS_14				: BYTE;									//{#lynus.ag#()}
	bySOC_E_CS_14			: BYTE;									//{#lynus.ag#()}
	bySOC_D_CS_14			: BYTE;									//{#lynus.ag#()}
	byMinPowerCS_14			: BYTE;									//{#lynus.ag#()}
	rMaxPowerCS_14			: REAL;									//{#lynus.ag#()}
	bEnabledCS_15			: BOOL;									//{#lynus.ag#()}
	byPrioCS_15				: BYTE;									//{#lynus.ag#()}
	bySOC_E_CS_15			: BYTE;									//{#lynus.ag#()}
	bySOC_D_CS_15			: BYTE;									//{#lynus.ag#()}
	byMinPowerCS_15			: BYTE;									//{#lynus.ag#()}
	rMaxPowerCS_15			: REAL;									//{#lynus.ag#()}
	bEnabledCS_16			: BOOL;									//{#lynus.ag#()}
	byPrioCS_16				: BYTE;									//{#lynus.ag#()}
	bySOC_E_CS_16			: BYTE;									//{#lynus.ag#()}
	bySOC_D_CS_16			: BYTE;									//{#lynus.ag#()}
	byMinPowerCS_16			: BYTE;									//{#lynus.ag#()}
	rMaxPowerCS_16			: REAL;									//{#lynus.ag#()}
	bEnabledCS_17			: BOOL;									//{#lynus.ag#()}
	byPrioCS_17				: BYTE;									//{#lynus.ag#()}
	bySOC_E_CS_17			: BYTE;									//{#lynus.ag#()}
	bySOC_D_CS_17			: BYTE;									//{#lynus.ag#()}
	byMinPowerCS_17			: BYTE;									//{#lynus.ag#()}
	rMaxPowerCS_17			: REAL;									//{#lynus.ag#()}
	bEnabledCS_18			: BOOL;									//{#lynus.ag#()}
	byPrioCS_18				: BYTE;									//{#lynus.ag#()}
	bySOC_E_CS_18			: BYTE;									//{#lynus.ag#()}
	bySOC_D_CS_18			: BYTE;									//{#lynus.ag#()}
	byMinPowerCS_18			: BYTE;									//{#lynus.ag#()}
	rMaxPowerCS_18			: REAL;									//{#lynus.ag#()}
END_VAR

// 10.10.122.101 Ladestation Gast LOW EWW
FB_KEBA_CS1(
	bEnable
	
FB_Schneider_EVLink_1(
	bEnable:= ,
	bEnableWrite:= TRUE , 
	bPowerDataInvers:= , 
	byElectricFuseLine:= , 
	rMinCurrent:= , 
	diNrOfEMS_IN:= prgEMS.fbEMS.diNrOfEMS_OUT,  
	diNrOfEM_IN_CS:= , 
	sIPAdress:= '10.10.122.101', 
	stSetupECS:= , 
	stDataECS=> , 
	diNrOfECS_OUT=> , 
	lrTotalPowerECSRealTime=> , 
	stDataElectric=> , 
	str_Mode3State=> , 
	bErrorCS=> , 
	lrTotalCounterEnergy_Consumption=> , 
	bCarConnected=> );
// 10.10.122.102 Ladestation Gast LOW EWW
FB_Schneider_EVLink_2(
	bEnable:= , 
	bEnableWrite:= TRUE, 
	bPowerDataInvers:= , 
	byElectricFuseLine:= , 
	rMinCurrent:= , 
	diNrOfEMS_IN:= prgEMS.fbEMS.diNrOfEMS_OUT,  
	diNrOfEM_IN_CS:= , 
	sIPAdress:=  '10.10.122.102', 
	stSetupECS:= , 
	stDataECS=> , 
	diNrOfECS_OUT=> , 
	lrTotalPowerECSRealTime=> , 
	stDataElectric=> , 
	str_Mode3State=> , 
	bErrorCS=> , 
	lrTotalCounterEnergy_Consumption=> , 
	bCarConnected=> );
	
// 10.10.122.103 Ladestation Intern Rechts LOW EWW
FB_Schneider_EVLink_3(
	bEnable:= , 
	bEnableWrite:= TRUE, 
	bPowerDataInvers:= , 
	byElectricFuseLine:= , 
	rMinCurrent:= , 
	diNrOfEMS_IN:= prgEMS.fbEMS.diNrOfEMS_OUT,  
	diNrOfEM_IN_CS:= , 
	sIPAdress:=  '10.10.122.103', 
	stSetupECS:= , 
	stDataECS=> , 
	diNrOfECS_OUT=> , 
	lrTotalPowerECSRealTime=> , 
	stDataElectric=> , 
	str_Mode3State=> , 
	bErrorCS=> , 
	lrTotalCounterEnergy_Consumption=> , 
	bCarConnected=> );
// 10.10.122.104 Ladestation Intern Rechts LOW EWW
FB_Schneider_EVLink_4(
	bEnable:= , 
	bEnableWrite:= TRUE, 
	bPowerDataInvers:= , 
	byElectricFuseLine:= , 
	rMinCurrent:= , 
	diNrOfEMS_IN:= prgEMS.fbEMS.diNrOfEMS_OUT,  
	diNrOfEM_IN_CS:= , 
	sIPAdress:=  '10.10.122.104', 
	stSetupECS:= , 
	stDataECS=> , 
	diNrOfECS_OUT=> , 
	lrTotalPowerECSRealTime=> , 
	stDataElectric=> , 
	str_Mode3State=> , 
	bErrorCS=> , 
	lrTotalCounterEnergy_Consumption=> , 
	bCarConnected=> );
// 10.10.122.105 Ladestation Intern Links LOW EWW
FB_Schneider_EVLink_5(
	bEnable:= , 
	bEnableWrite:= TRUE, 
	bPowerDataInvers:= , 
	byElectricFuseLine:= , 
	rMinCurrent:= , 
	diNrOfEMS_IN:= prgEMS.fbEMS.diNrOfEMS_OUT,  
	diNrOfEM_IN_CS:= , 
	sIPAdress:=  '10.10.122.105', 
	stSetupECS:= , 
	stDataECS=> , 
	diNrOfECS_OUT=> , 
	lrTotalPowerECSRealTime=> , 
	stDataElectric=> , 
	str_Mode3State=> , 
	bErrorCS=> , 
	lrTotalCounterEnergy_Consumption=> , 
	bCarConnected=> );
// 10.10.122.106 Ladestation Intern Links LOW EWW
FB_Schneider_EVLink_6(
	bEnable:= , 
	bEnableWrite:= TRUE , 
	bPowerDataInvers:= , 
	byElectricFuseLine:= , 
	rMinCurrent:= , 
	diNrOfEMS_IN:= prgEMS.fbEMS.diNrOfEMS_OUT,  
	diNrOfEM_IN_CS:= , 
	sIPAdress:=  '10.10.122.106', 
	stSetupECS:= , 
	stDataECS=> , 
	diNrOfECS_OUT=> , 
	lrTotalPowerECSRealTime=> , 
	stDataElectric=> , 
	str_Mode3State=> , 
	bErrorCS=> , 
	lrTotalCounterEnergy_Consumption=> , 
	bCarConnected=> );
// 10.10.122.113 Ladestation Neu 1 LOW Ladestation Intern1 Links
FB_Schneider_EVLink_7(
	bEnable:= , 
	bEnableWrite:= TRUE, 
	bPowerDataInvers:= , 
	byElectricFuseLine:= , 
	rMinCurrent:= , 
	diNrOfEMS_IN:= prgEMS.fbEMS.diNrOfEMS_OUT,  
	diNrOfEM_IN_CS:= , 
	sIPAdress:=  '10.10.122.113', 
	stSetupECS:= , 
	stDataECS=> , 
	diNrOfECS_OUT=> , 
	lrTotalPowerECSRealTime=> , 
	stDataElectric=> , 
	str_Mode3State=> , 
	bErrorCS=> , 
	lrTotalCounterEnergy_Consumption=> , 
	bCarConnected=> );
// 10.10.122.114 Ladestation Neu 2 LOW
FB_Schneider_EVLink_8(
	bEnable:= , 
	bEnableWrite:= TRUE , 
	bPowerDataInvers:= , 
	byElectricFuseLine:= , 
	rMinCurrent:= , 
	diNrOfEMS_IN:= prgEMS.fbEMS.diNrOfEMS_OUT,  
	diNrOfEM_IN_CS:= , 
	sIPAdress:=  '10.10.122.114', 
	stSetupECS:= , 
	stDataECS=> , 
	diNrOfECS_OUT=> , 
	lrTotalPowerECSRealTime=> , 
	stDataElectric=> , 
	str_Mode3State=> , 
	bErrorCS=> , 
	lrTotalCounterEnergy_Consumption=> , 
	bCarConnected=> );
// 10.10.122.115 Ladestation Neu 3 LOW Ladestation Intern1 Mitte
FB_Schneider_EVLink_9(
	bEnable:= , 
	bEnableWrite:= TRUE , 
	bPowerDataInvers:= , 
	byElectricFuseLine:= , 
	rMinCurrent:= , 
	diNrOfEMS_IN:= prgEMS.fbEMS.diNrOfEMS_OUT,  
	diNrOfEM_IN_CS:= , 
	sIPAdress:=  '10.10.122.115', 
	stSetupECS:= , 
	stDataECS=> , 
	diNrOfECS_OUT=> , 
	lrTotalPowerECSRealTime=> , 
	stDataElectric=> , 
	str_Mode3State=> , 
	bErrorCS=> , 
	lrTotalCounterEnergy_Consumption=> , 
	bCarConnected=> );
// 10.10.122.116 Ladestation Neu 4 LOW
FB_Schneider_EVLink_10(
	bEnable:= , 
	bEnableWrite:= TRUE, 
	bPowerDataInvers:= , 
	byElectricFuseLine:= , 
	rMinCurrent:= , 
	diNrOfEMS_IN:= prgEMS.fbEMS.diNrOfEMS_OUT,  
	diNrOfEM_IN_CS:= , 
	sIPAdress:=  '10.10.122.116', 
	stSetupECS:= , 
	stDataECS=> , 
	diNrOfECS_OUT=> , 
	lrTotalPowerECSRealTime=> , 
	stDataElectric=> , 
	str_Mode3State=> , 
	bErrorCS=> , 
	lrTotalCounterEnergy_Consumption=> , 
	bCarConnected=> );
// 10.10.122.117 Ladestation Neu 5 LOW Ladestation Intern2 Rechts
FB_Schneider_EVLink_11(
	bEnable:= , 
	bEnableWrite:= TRUE, 
	bPowerDataInvers:= , 
	byElectricFuseLine:= , 
	rMinCurrent:= , 
	diNrOfEMS_IN:= prgEMS.fbEMS.diNrOfEMS_OUT,  
	diNrOfEM_IN_CS:= , 
	sIPAdress:=  '10.10.122.117', 
	stSetupECS:= , 
	stDataECS=> , 
	diNrOfECS_OUT=> , 
	lrTotalPowerECSRealTime=> , 
	stDataElectric=> , 
	str_Mode3State=> , 
	bErrorCS=> , 
	lrTotalCounterEnergy_Consumption=> , 
	bCarConnected=> );
// 10.10.122.118 Ladestation Neu 6 LOW
FB_Schneider_EVLink_12(
	bEnable:= , 
	bEnableWrite:= TRUE, 
	bPowerDataInvers:= , 
	byElectricFuseLine:= , 
	rMinCurrent:= , 
	diNrOfEMS_IN:= prgEMS.fbEMS.diNrOfEMS_OUT,  
	diNrOfEM_IN_CS:= , 
	sIPAdress:=  '10.10.122.118', 
	stSetupECS:= , 
	stDataECS=> , 
	diNrOfECS_OUT=> , 
	lrTotalPowerECSRealTime=> , 
	stDataElectric=> , 
	str_Mode3State=> , 
	bErrorCS=> , 
	lrTotalCounterEnergy_Consumption=> , 
	bCarConnected=> );
// 10.10.122.119 Ladestation Neu 7 LOW Ladestation Intern2 Links
FB_Schneider_EVLink_13(
	bEnable:= , 
	bEnableWrite:= TRUE, 
	bPowerDataInvers:= , 
	byElectricFuseLine:= , 
	rMinCurrent:= , 
	diNrOfEMS_IN:= prgEMS.fbEMS.diNrOfEMS_OUT,  
	diNrOfEM_IN_CS:= , 
	sIPAdress:=  '10.10.122.119', 
	stSetupECS:= , 
	stDataECS=> , 
	diNrOfECS_OUT=> , 
	lrTotalPowerECSRealTime=> , 
	stDataElectric=> , 
	str_Mode3State=> , 
	bErrorCS=> , 
	lrTotalCounterEnergy_Consumption=> , 
	bCarConnected=> );
// 10.10.122.120 Ladestation Neu 8 LOW
FB_Schneider_EVLink_14(
	bEnable:= , 
	bEnableWrite:= TRUE, 
	bPowerDataInvers:= , 
	byElectricFuseLine:= , 
	rMinCurrent:= , 
	diNrOfEMS_IN:= prgEMS.fbEMS.diNrOfEMS_OUT,  
	diNrOfEM_IN_CS:= , 
	sIPAdress:=  '10.10.122.120', 
	stSetupECS:= , 
	stDataECS=> , 
	diNrOfECS_OUT=> , 
	lrTotalPowerECSRealTime=> , 
	stDataElectric=> , 
	str_Mode3State=> , 
	bErrorCS=> , 
	lrTotalCounterEnergy_Consumption=> , 
	bCarConnected=> );
// 10.10.122.121 Ladestation Neu 9 LOW
FB_Schneider_EVLink_15(
	bEnable:= , 
	bEnableWrite:= TRUE, 
	bPowerDataInvers:= , 
	byElectricFuseLine:= , 
	rMinCurrent:= , 
	diNrOfEMS_IN:= prgEMS.fbEMS.diNrOfEMS_OUT,  
	diNrOfEM_IN_CS:= , 
	sIPAdress:=  '10.10.122.121', 
	stSetupECS:= , 
	stDataECS=> , 
	diNrOfECS_OUT=> , 
	lrTotalPowerECSRealTime=> , 
	stDataElectric=> , 
	str_Mode3State=> , 
	bErrorCS=> , 
	lrTotalCounterEnergy_Consumption=> , 
	bCarConnected=> );
// 10.10.122.122 Ladestation Neu 10 LOW
FB_Schneider_EVLink_16(
	bEnable:= , 
	bEnableWrite:= TRUE, 
	bPowerDataInvers:= , 
	byElectricFuseLine:= , 
	rMinCurrent:= , 
	diNrOfEMS_IN:= prgEMS.fbEMS.diNrOfEMS_OUT,  
	diNrOfEM_IN_CS:= , 
	sIPAdress:=  '10.10.122.122', 
	stSetupECS:= , 
	stDataECS=> , 
	diNrOfECS_OUT=> , 
	lrTotalPowerECSRealTime=> , 
	stDataElectric=> , 
	str_Mode3State=> , 
	bErrorCS=> , 
	lrTotalCounterEnergy_Consumption=> , 
	bCarConnected=> );
// 10.10.122.123 Ladestation Neu 11 LOW
FB_Schneider_EVLink_17(
	bEnable:= , 
	bEnableWrite:= TRUE, 
	bPowerDataInvers:= , 
	byElectricFuseLine:= , 
	rMinCurrent:= , 
	diNrOfEMS_IN:= prgEMS.fbEMS.diNrOfEMS_OUT,  
	diNrOfEM_IN_CS:= , 
	sIPAdress:=  '10.10.122.123', 
	stSetupECS:= , 
	stDataECS=> , 
	diNrOfECS_OUT=> , 
	lrTotalPowerECSRealTime=> , 
	stDataElectric=> , 
	str_Mode3State=> , 
	bErrorCS=> , 
	lrTotalCounterEnergy_Consumption=> , 
	bCarConnected=> );
// 10.10.122.124 Ladestation Neu 12 LOW
FB_Schneider_EVLink_18(
	bEnable:= , 
	bEnableWrite:= TRUE , 
	bPowerDataInvers:= , 
	byElectricFuseLine:= , 
	rMinCurrent:= , 
	diNrOfEMS_IN:= prgEMS.fbEMS.diNrOfEMS_OUT,  
	diNrOfEM_IN_CS:= , 
	sIPAdress:=  '10.10.122.124', 
	stSetupECS:= , 
	stDataECS=> , 
	diNrOfECS_OUT=> , 
	lrTotalPowerECSRealTime=> , 
	stDataElectric=> , 
	str_Mode3State=> , 
	bErrorCS=> , 
	lrTotalCounterEnergy_Consumption=> , 
	bCarConnected=> );

	
lr_CSPowerTotal :=	FB_Schneider_EVLink_1.stDataElectric.lrPowerTotal + FB_Schneider_EVLink_2.stDataElectric.lrPowerTotal + FB_Schneider_EVLink_3.stDataElectric.lrPowerTotal + 
				FB_Schneider_EVLink_4.stDataElectric.lrPowerTotal + FB_Schneider_EVLink_5.stDataElectric.lrPowerTotal + FB_Schneider_EVLink_6.stDataElectric.lrPowerTotal +
				FB_Schneider_EVLink_7.stDataElectric.lrPowerTotal + FB_Schneider_EVLink_8.stDataElectric.lrPowerTotal + FB_Schneider_EVLink_9.stDataElectric.lrPowerTotal +  
				FB_Schneider_EVLink_10.stDataElectric.lrPowerTotal + FB_Schneider_EVLink_11.stDataElectric.lrPowerTotal + FB_Schneider_EVLink_12.stDataElectric.lrPowerTotal +
				FB_Schneider_EVLink_13.stDataElectric.lrPowerTotal + FB_Schneider_EVLink_14.stDataElectric.lrPowerTotal + FB_Schneider_EVLink_15.stDataElectric.lrPowerTotal +
				FB_Schneider_EVLink_16.stDataElectric.lrPowerTotal + FB_Schneider_EVLink_17.stDataElectric.lrPowerTotal + FB_Schneider_EVLink_18.stDataElectric.lrPowerTotal;

lr_CSEnergy_Total := FB_Schneider_EVLink_1.lrTotalCounterEnergy_Consumption + FB_Schneider_EVLink_2.lrTotalCounterEnergy_Consumption + FB_Schneider_EVLink_3.lrTotalCounterEnergy_Consumption + 
				FB_Schneider_EVLink_4.lrTotalCounterEnergy_Consumption + FB_Schneider_EVLink_5.lrTotalCounterEnergy_Consumption + FB_Schneider_EVLink_6.lrTotalCounterEnergy_Consumption +
				FB_Schneider_EVLink_7.lrTotalCounterEnergy_Consumption + FB_Schneider_EVLink_8.lrTotalCounterEnergy_Consumption + FB_Schneider_EVLink_9.lrTotalCounterEnergy_Consumption +  
				FB_Schneider_EVLink_10.lrTotalCounterEnergy_Consumption + FB_Schneider_EVLink_11.lrTotalCounterEnergy_Consumption + FB_Schneider_EVLink_12.lrTotalCounterEnergy_Consumption +
				FB_Schneider_EVLink_13.lrTotalCounterEnergy_Consumption + FB_Schneider_EVLink_14.lrTotalCounterEnergy_Consumption + FB_Schneider_EVLink_15.lrTotalCounterEnergy_Consumption +
				FB_Schneider_EVLink_16.lrTotalCounterEnergy_Consumption + FB_Schneider_EVLink_17.lrTotalCounterEnergy_Consumption + FB_Schneider_EVLink_18.lrTotalCounterEnergy_Consumption;
	
FB_Schneider_EVLink_1.stSetupECS.byDisableSOC 	:= bySOC_D_CS_1;		   			
FB_Schneider_EVLink_1.stSetupECS.byEnableSOC 	:= bySOC_E_CS_1;	
FB_Schneider_EVLink_1.stSetupECS.byPriority 	:= byPrioCS_1;
FB_Schneider_EVLink_1.stSetupECS.rMaxPower 		:= rMaxPowerCS_1;
FB_Schneider_EVLink_1.stSetupECS.byCSMinPower	:= byMinPowerCS_1;
FB_Schneider_EVLink_1.bEnable					:= bEnabledCS_1;
FB_Schneider_EVLink_1.stSetupECS.bManualyOn		:= bChrgManuCS_1;
FB_Schneider_EVLink_1.stSetupECS.byManualyTargetPower := byChrgManuSPCS_1;

bIsEnabledCS_1 		:= FB_Schneider_EVLink_1.stDataECS.bEnabled;
byStateMinPowerCS_1 := FB_Schneider_EVLink_1.stDataECS.bySCSMinPower;
rTargetPowerCS_1 	:= FB_Schneider_EVLink_1.stDataECS.rTargetPower;	
byErrorWarningCS_1 	:= FB_Schneider_EVLink_1.stDataECS.byErrorWarning;
bCarConnectedCS_1 	:= FB_Schneider_EVLink_1.stDataECS.bCarConnected;
rChrgTimeCS_1 		:= FB_Schneider_EVLink_1.stDataECS.arrChargingTimeInMin[1];
lr_CSPower_1 		:= FB_Schneider_EVLink_1.stDataElectric.lrPowerTotal;
bStateOkCS_1		:= FB_Schneider_EVLink_1.bEnable AND FB_Schneider_EVLink_1.bEnableWrite;

FB_Schneider_EVLink_2.stSetupECS.byDisableSOC 	:= bySOC_D_CS_2;		   			
FB_Schneider_EVLink_2.stSetupECS.byEnableSOC 	:= bySOC_E_CS_2;	
FB_Schneider_EVLink_2.stSetupECS.byPriority 	:= byPrioCS_2;
FB_Schneider_EVLink_2.stSetupECS.rMaxPower 		:= rMaxPowerCS_2;
FB_Schneider_EVLink_2.stSetupECS.byCSMinPower	:= byMinPowerCS_2;
FB_Schneider_EVLink_2.bEnable					:= bEnabledCS_2;
FB_Schneider_EVLink_2.stSetupECS.bManualyOn		:= bChrgManuCS_2;
FB_Schneider_EVLink_2.stSetupECS.byManualyTargetPower := byChrgManuSPCS_2;

bIsEnabledCS_2 		:= FB_Schneider_EVLink_2.stDataECS.bEnabled;
byStateMinPowerCS_2 := FB_Schneider_EVLink_2.stDataECS.bySCSMinPower;
rTargetPowerCS_2 	:= FB_Schneider_EVLink_2.stDataECS.rTargetPower;	
byErrorWarningCS_2 	:= FB_Schneider_EVLink_2.stDataECS.byErrorWarning;
bCarConnectedCS_2 	:= FB_Schneider_EVLink_2.stDataECS.bCarConnected;
rChrgTimeCS_2 		:= FB_Schneider_EVLink_2.stDataECS.arrChargingTimeInMin[1];
lr_CSPower_2 		:= FB_Schneider_EVLink_2.stDataElectric.lrPowerTotal;
bStateOkCS_2		:= FB_Schneider_EVLink_2.bEnable AND FB_Schneider_EVLink_2.bEnableWrite;

FB_Schneider_EVLink_3.stSetupECS.byDisableSOC 	:= bySOC_D_CS_3;		   			
FB_Schneider_EVLink_3.stSetupECS.byEnableSOC 	:= bySOC_E_CS_3;	
FB_Schneider_EVLink_3.stSetupECS.byPriority 	:= byPrioCS_3;
FB_Schneider_EVLink_3.stSetupECS.rMaxPower 		:= rMaxPowerCS_3;
FB_Schneider_EVLink_3.stSetupECS.byCSMinPower	:= byMinPowerCS_3;
FB_Schneider_EVLink_3.bEnable					:= bEnabledCS_3;
FB_Schneider_EVLink_3.stSetupECS.bManualyOn		:= bChrgManuCS_3;
FB_Schneider_EVLink_3.stSetupECS.byManualyTargetPower := byChrgManuSPCS_3;

bIsEnabledCS_3 		:= FB_Schneider_EVLink_3.stDataECS.bEnabled;
byStateMinPowerCS_3 := FB_Schneider_EVLink_3.stDataECS.bySCSMinPower;
rTargetPowerCS_3 	:= FB_Schneider_EVLink_3.stDataECS.rTargetPower;	
byErrorWarningCS_3 	:= FB_Schneider_EVLink_3.stDataECS.byErrorWarning;
bCarConnectedCS_3 	:= FB_Schneider_EVLink_3.stDataECS.bCarConnected;
rChrgTimeCS_3 		:= FB_Schneider_EVLink_3.stDataECS.arrChargingTimeInMin[1];
lr_CSPower_3 		:= FB_Schneider_EVLink_3.stDataElectric.lrPowerTotal;
bStateOkCS_3		:= FB_Schneider_EVLink_3.bEnable AND FB_Schneider_EVLink_3.bEnableWrite;


FB_Schneider_EVLink_4.stSetupECS.byDisableSOC 	:= bySOC_D_CS_4;		   			
FB_Schneider_EVLink_4.stSetupECS.byEnableSOC 	:= bySOC_E_CS_4;	
FB_Schneider_EVLink_4.stSetupECS.byPriority 	:= byPrioCS_4;
FB_Schneider_EVLink_4.stSetupECS.rMaxPower 		:= rMaxPowerCS_4;
FB_Schneider_EVLink_4.stSetupECS.byCSMinPower	:= byMinPowerCS_4;
FB_Schneider_EVLink_4.bEnable					:= bEnabledCS_4;
FB_Schneider_EVLink_4.stSetupECS.bManualyOn		:= bChrgManuCS_4;
FB_Schneider_EVLink_4.stSetupECS.byManualyTargetPower := byChrgManuSPCS_4;

bIsEnabledCS_4 		:= FB_Schneider_EVLink_4.stDataECS.bEnabled;
byStateMinPowerCS_4 := FB_Schneider_EVLink_4.stDataECS.bySCSMinPower;
rTargetPowerCS_4 	:= FB_Schneider_EVLink_4.stDataECS.rTargetPower;	
byErrorWarningCS_4 	:= FB_Schneider_EVLink_4.stDataECS.byErrorWarning;
bCarConnectedCS_4 	:= FB_Schneider_EVLink_4.stDataECS.bCarConnected;
rChrgTimeCS_4 		:= FB_Schneider_EVLink_4.stDataECS.arrChargingTimeInMin[1];
lr_CSPower_4 		:= FB_Schneider_EVLink_4.stDataElectric.lrPowerTotal;
bStateOkCS_4		:= FB_Schneider_EVLink_4.bEnable AND FB_Schneider_EVLink_4.bEnableWrite;


FB_Schneider_EVLink_5.stSetupECS.byDisableSOC 	:= bySOC_D_CS_5;		   			
FB_Schneider_EVLink_5.stSetupECS.byEnableSOC 	:= bySOC_E_CS_5;	
FB_Schneider_EVLink_5.stSetupECS.byPriority 	:= byPrioCS_5;
FB_Schneider_EVLink_5.stSetupECS.rMaxPower 		:= rMaxPowerCS_5;
FB_Schneider_EVLink_5.stSetupECS.byCSMinPower	:= byMinPowerCS_5;
FB_Schneider_EVLink_5.bEnable					:= bEnabledCS_5;
FB_Schneider_EVLink_5.stSetupECS.bManualyOn		:= bChrgManuCS_5;
FB_Schneider_EVLink_5.stSetupECS.byManualyTargetPower := byChrgManuSPCS_5;

bIsEnabledCS_5 		:= FB_Schneider_EVLink_5.stDataECS.bEnabled;
byStateMinPowerCS_5 := FB_Schneider_EVLink_5.stDataECS.bySCSMinPower;
rTargetPowerCS_5 	:= FB_Schneider_EVLink_5.stDataECS.rTargetPower;	
byErrorWarningCS_5 	:= FB_Schneider_EVLink_5.stDataECS.byErrorWarning;
bCarConnectedCS_5 	:= FB_Schneider_EVLink_5.stDataECS.bCarConnected;
rChrgTimeCS_5 		:= FB_Schneider_EVLink_5.stDataECS.arrChargingTimeInMin[1];
lr_CSPower_5 		:= FB_Schneider_EVLink_5.stDataElectric.lrPowerTotal;
bStateOkCS_5		:= FB_Schneider_EVLink_5.bEnable AND FB_Schneider_EVLink_5.bEnableWrite;


FB_Schneider_EVLink_6.stSetupECS.byDisableSOC 	:= bySOC_D_CS_6;		   			
FB_Schneider_EVLink_6.stSetupECS.byEnableSOC 	:= bySOC_E_CS_6;	
FB_Schneider_EVLink_6.stSetupECS.byPriority 	:= byPrioCS_6;
FB_Schneider_EVLink_6.stSetupECS.rMaxPower 		:= rMaxPowerCS_6;
FB_Schneider_EVLink_6.stSetupECS.byCSMinPower	:= byMinPowerCS_6;
FB_Schneider_EVLink_6.bEnable					:= bEnabledCS_6;
FB_Schneider_EVLink_6.stSetupECS.bManualyOn		:= bChrgManuCS_6;
FB_Schneider_EVLink_6.stSetupECS.byManualyTargetPower := byChrgManuSPCS_6;

bIsEnabledCS_6 		:= FB_Schneider_EVLink_6.stDataECS.bEnabled;
byStateMinPowerCS_6 := FB_Schneider_EVLink_6.stDataECS.bySCSMinPower;
rTargetPowerCS_6 	:= FB_Schneider_EVLink_6.stDataECS.rTargetPower;	
byErrorWarningCS_6 	:= FB_Schneider_EVLink_6.stDataECS.byErrorWarning;
bCarConnectedCS_6 	:= FB_Schneider_EVLink_6.stDataECS.bCarConnected;
rChrgTimeCS_6 		:= FB_Schneider_EVLink_6.stDataECS.arrChargingTimeInMin[1];
lr_CSPower_6 		:= FB_Schneider_EVLink_6.stDataElectric.lrPowerTotal;
bStateOkCS_6		:= FB_Schneider_EVLink_6.bEnable AND FB_Schneider_EVLink_6.bEnableWrite;

FB_Schneider_EVLink_7.stSetupECS.byDisableSOC 	:= bySOC_D_CS_7;		   			
FB_Schneider_EVLink_7.stSetupECS.byEnableSOC 	:= bySOC_E_CS_7;	
FB_Schneider_EVLink_7.stSetupECS.byPriority 	:= byPrioCS_7;
FB_Schneider_EVLink_7.stSetupECS.rMaxPower 		:= rMaxPowerCS_7;
FB_Schneider_EVLink_7.stSetupECS.byCSMinPower	:= byMinPowerCS_7;
FB_Schneider_EVLink_7.bEnable					:= bEnabledCS_7;
FB_Schneider_EVLink_7.stSetupECS.bManualyOn		:= bChrgManuCS_7;
FB_Schneider_EVLink_7.stSetupECS.byManualyTargetPower := byChrgManuSPCS_7;

bIsEnabledCS_7 		:= FB_Schneider_EVLink_7.stDataECS.bEnabled;
byStateMinPowerCS_7 := FB_Schneider_EVLink_7.stDataECS.bySCSMinPower;
rTargetPowerCS_7 	:= FB_Schneider_EVLink_7.stDataECS.rTargetPower;	
byErrorWarningCS_7 	:= FB_Schneider_EVLink_7.stDataECS.byErrorWarning;
bCarConnectedCS_7 	:= FB_Schneider_EVLink_7.stDataECS.bCarConnected;
rChrgTimeCS_7 		:= FB_Schneider_EVLink_7.stDataECS.arrChargingTimeInMin[1];
lr_CSPower_7 		:= FB_Schneider_EVLink_7.stDataElectric.lrPowerTotal;
bStateOkCS_7		:= FB_Schneider_EVLink_7.bEnable AND FB_Schneider_EVLink_7.bEnableWrite;

FB_Schneider_EVLink_8.stSetupECS.byDisableSOC 	:= bySOC_D_CS_8;		   			
FB_Schneider_EVLink_8.stSetupECS.byEnableSOC 	:= bySOC_E_CS_8;	
FB_Schneider_EVLink_8.stSetupECS.byPriority 	:= byPrioCS_8;
FB_Schneider_EVLink_8.stSetupECS.rMaxPower 		:= rMaxPowerCS_8;
FB_Schneider_EVLink_8.stSetupECS.byCSMinPower	:= byMinPowerCS_8;
FB_Schneider_EVLink_8.bEnable					:= bEnabledCS_8;
FB_Schneider_EVLink_8.stSetupECS.bManualyOn		:= bChrgManuCS_8;
FB_Schneider_EVLink_8.stSetupECS.byManualyTargetPower := byChrgManuSPCS_8;

bIsEnabledCS_8 		:= FB_Schneider_EVLink_8.stDataECS.bEnabled;
byStateMinPowerCS_8 := FB_Schneider_EVLink_8.stDataECS.bySCSMinPower;
rTargetPowerCS_8 	:= FB_Schneider_EVLink_8.stDataECS.rTargetPower;	
byErrorWarningCS_8 	:= FB_Schneider_EVLink_8.stDataECS.byErrorWarning;
bCarConnectedCS_8 	:= FB_Schneider_EVLink_8.stDataECS.bCarConnected;
rChrgTimeCS_8 		:= FB_Schneider_EVLink_8.stDataECS.arrChargingTimeInMin[1];
lr_CSPower_8 		:= FB_Schneider_EVLink_8.stDataElectric.lrPowerTotal;
bStateOkCS_8		:= FB_Schneider_EVLink_8.bEnable AND FB_Schneider_EVLink_8.bEnableWrite;

FB_Schneider_EVLink_9.stSetupECS.byDisableSOC 	:= bySOC_D_CS_9;		   			
FB_Schneider_EVLink_9.stSetupECS.byEnableSOC 	:= bySOC_E_CS_9;	
FB_Schneider_EVLink_9.stSetupECS.byPriority 	:= byPrioCS_9;
FB_Schneider_EVLink_9.stSetupECS.rMaxPower 		:= rMaxPowerCS_9;
FB_Schneider_EVLink_9.stSetupECS.byCSMinPower	:= byMinPowerCS_9;
FB_Schneider_EVLink_9.bEnable					:= bEnabledCS_9;
FB_Schneider_EVLink_9.stSetupECS.bManualyOn		:= bChrgManuCS_9;
FB_Schneider_EVLink_9.stSetupECS.byManualyTargetPower := byChrgManuSPCS_9;

bIsEnabledCS_9 		:= FB_Schneider_EVLink_9.stDataECS.bEnabled;
byStateMinPowerCS_9 := FB_Schneider_EVLink_9.stDataECS.bySCSMinPower;
rTargetPowerCS_9 	:= FB_Schneider_EVLink_9.stDataECS.rTargetPower;	
byErrorWarningCS_9 	:= FB_Schneider_EVLink_9.stDataECS.byErrorWarning;
bCarConnectedCS_9 	:= FB_Schneider_EVLink_9.stDataECS.bCarConnected;
rChrgTimeCS_9 		:= FB_Schneider_EVLink_9.stDataECS.arrChargingTimeInMin[1];
lr_CSPower_9 		:= FB_Schneider_EVLink_9.stDataElectric.lrPowerTotal;
bStateOkCS_9		:= FB_Schneider_EVLink_9.bEnable AND FB_Schneider_EVLink_9.bEnableWrite;


FB_Schneider_EVLink_10.stSetupECS.byDisableSOC 	:= bySOC_D_CS_10;		   			
FB_Schneider_EVLink_10.stSetupECS.byEnableSOC 	:= bySOC_E_CS_10;	
FB_Schneider_EVLink_10.stSetupECS.byPriority 	:= byPrioCS_10;
FB_Schneider_EVLink_10.stSetupECS.rMaxPower 		:= rMaxPowerCS_10;
FB_Schneider_EVLink_10.stSetupECS.byCSMinPower	:= byMinPowerCS_10;
FB_Schneider_EVLink_10.bEnable					:= bEnabledCS_10;
FB_Schneider_EVLink_10.stSetupECS.bManualyOn		:= bChrgManuCS_10;
FB_Schneider_EVLink_10.stSetupECS.byManualyTargetPower := byChrgManuSPCS_10;

bIsEnabledCS_10 		:= FB_Schneider_EVLink_10.stDataECS.bEnabled;
byStateMinPowerCS_10 := FB_Schneider_EVLink_10.stDataECS.bySCSMinPower;
rTargetPowerCS_10 	:= FB_Schneider_EVLink_10.stDataECS.rTargetPower;	
byErrorWarningCS_10 	:= FB_Schneider_EVLink_10.stDataECS.byErrorWarning;
bCarConnectedCS_10 	:= FB_Schneider_EVLink_10.stDataECS.bCarConnected;
rChrgTimeCS_10 		:= FB_Schneider_EVLink_10.stDataECS.arrChargingTimeInMin[1];
lr_CSPower_10 		:= FB_Schneider_EVLink_10.stDataElectric.lrPowerTotal;
bStateOkCS_10		:= FB_Schneider_EVLink_10.bEnable AND FB_Schneider_EVLink_10.bEnableWrite;

FB_Schneider_EVLink_11.stSetupECS.byDisableSOC 	:= bySOC_D_CS_11;		   			
FB_Schneider_EVLink_11.stSetupECS.byEnableSOC 	:= bySOC_E_CS_11;	
FB_Schneider_EVLink_11.stSetupECS.byPriority 	:= byPrioCS_11;
FB_Schneider_EVLink_11.stSetupECS.rMaxPower 		:= rMaxPowerCS_11;
FB_Schneider_EVLink_11.stSetupECS.byCSMinPower	:= byMinPowerCS_11;
FB_Schneider_EVLink_11.bEnable					:= bEnabledCS_11;
FB_Schneider_EVLink_11.stSetupECS.bManualyOn		:= bChrgManuCS_11;
FB_Schneider_EVLink_11.stSetupECS.byManualyTargetPower := byChrgManuSPCS_11;

bIsEnabledCS_11 		:= FB_Schneider_EVLink_11.stDataECS.bEnabled;
byStateMinPowerCS_11 := FB_Schneider_EVLink_11.stDataECS.bySCSMinPower;
rTargetPowerCS_11 	:= FB_Schneider_EVLink_11.stDataECS.rTargetPower;	
byErrorWarningCS_11 	:= FB_Schneider_EVLink_11.stDataECS.byErrorWarning;
bCarConnectedCS_11 	:= FB_Schneider_EVLink_11.stDataECS.bCarConnected;
rChrgTimeCS_11 		:= FB_Schneider_EVLink_11.stDataECS.arrChargingTimeInMin[1];
lr_CSPower_11 		:= FB_Schneider_EVLink_11.stDataElectric.lrPowerTotal;
bStateOkCS_11		:= FB_Schneider_EVLink_11.bEnable AND FB_Schneider_EVLink_11.bEnableWrite;

FB_Schneider_EVLink_12.stSetupECS.byDisableSOC 	:= bySOC_D_CS_12;		   			
FB_Schneider_EVLink_12.stSetupECS.byEnableSOC 	:= bySOC_E_CS_12;	
FB_Schneider_EVLink_12.stSetupECS.byPriority 	:= byPrioCS_12;
FB_Schneider_EVLink_12.stSetupECS.rMaxPower 		:= rMaxPowerCS_12;
FB_Schneider_EVLink_12.stSetupECS.byCSMinPower	:= byMinPowerCS_12;
FB_Schneider_EVLink_12.bEnable					:= bEnabledCS_12;
FB_Schneider_EVLink_12.stSetupECS.bManualyOn		:= bChrgManuCS_12;
FB_Schneider_EVLink_12.stSetupECS.byManualyTargetPower := byChrgManuSPCS_12;

bIsEnabledCS_12 		:= FB_Schneider_EVLink_12.stDataECS.bEnabled;
byStateMinPowerCS_12 := FB_Schneider_EVLink_12.stDataECS.bySCSMinPower;
rTargetPowerCS_12 	:= FB_Schneider_EVLink_12.stDataECS.rTargetPower;	
byErrorWarningCS_12 	:= FB_Schneider_EVLink_12.stDataECS.byErrorWarning;
bCarConnectedCS_12 	:= FB_Schneider_EVLink_12.stDataECS.bCarConnected;
rChrgTimeCS_12 		:= FB_Schneider_EVLink_12.stDataECS.arrChargingTimeInMin[1];
lr_CSPower_12 		:= FB_Schneider_EVLink_12.stDataElectric.lrPowerTotal;
bStateOkCS_12		:= FB_Schneider_EVLink_12.bEnable AND FB_Schneider_EVLink_12.bEnableWrite;

FB_Schneider_EVLink_13.stSetupECS.byDisableSOC 	:= bySOC_D_CS_13;		   			
FB_Schneider_EVLink_13.stSetupECS.byEnableSOC 	:= bySOC_E_CS_13;	
FB_Schneider_EVLink_13.stSetupECS.byPriority 	:= byPrioCS_13;
FB_Schneider_EVLink_13.stSetupECS.rMaxPower 		:= rMaxPowerCS_13;
FB_Schneider_EVLink_13.stSetupECS.byCSMinPower	:= byMinPowerCS_13;
FB_Schneider_EVLink_13.bEnable					:= bEnabledCS_13;
FB_Schneider_EVLink_13.stSetupECS.bManualyOn		:= bChrgManuCS_13;
FB_Schneider_EVLink_13.stSetupECS.byManualyTargetPower := byChrgManuSPCS_13;

bIsEnabledCS_13 		:= FB_Schneider_EVLink_13.stDataECS.bEnabled;
byStateMinPowerCS_13 := FB_Schneider_EVLink_13.stDataECS.bySCSMinPower;
rTargetPowerCS_13 	:= FB_Schneider_EVLink_13.stDataECS.rTargetPower;	
byErrorWarningCS_13 	:= FB_Schneider_EVLink_13.stDataECS.byErrorWarning;
bCarConnectedCS_13 	:= FB_Schneider_EVLink_13.stDataECS.bCarConnected;
rChrgTimeCS_13 		:= FB_Schneider_EVLink_13.stDataECS.arrChargingTimeInMin[1];
lr_CSPower_13 		:= FB_Schneider_EVLink_13.stDataElectric.lrPowerTotal;
bStateOkCS_13		:= FB_Schneider_EVLink_13.bEnable AND FB_Schneider_EVLink_13.bEnableWrite;

FB_Schneider_EVLink_14.stSetupECS.byDisableSOC 	:= bySOC_D_CS_14;		   			
FB_Schneider_EVLink_14.stSetupECS.byEnableSOC 	:= bySOC_E_CS_14;	
FB_Schneider_EVLink_14.stSetupECS.byPriority 	:= byPrioCS_14;
FB_Schneider_EVLink_14.stSetupECS.rMaxPower 		:= rMaxPowerCS_14;
FB_Schneider_EVLink_14.stSetupECS.byCSMinPower	:= byMinPowerCS_14;
FB_Schneider_EVLink_14.bEnable					:= bEnabledCS_14;
FB_Schneider_EVLink_14.stSetupECS.bManualyOn		:= bChrgManuCS_14;
FB_Schneider_EVLink_14.stSetupECS.byManualyTargetPower := byChrgManuSPCS_14;

bIsEnabledCS_14 		:= FB_Schneider_EVLink_14.stDataECS.bEnabled;
byStateMinPowerCS_14 := FB_Schneider_EVLink_14.stDataECS.bySCSMinPower;
rTargetPowerCS_14 	:= FB_Schneider_EVLink_14.stDataECS.rTargetPower;	
byErrorWarningCS_14 	:= FB_Schneider_EVLink_14.stDataECS.byErrorWarning;
bCarConnectedCS_14 	:= FB_Schneider_EVLink_14.stDataECS.bCarConnected;
rChrgTimeCS_14 		:= FB_Schneider_EVLink_14.stDataECS.arrChargingTimeInMin[1];
lr_CSPower_14 		:= FB_Schneider_EVLink_14.stDataElectric.lrPowerTotal;
bStateOkCS_14		:= FB_Schneider_EVLink_14.bEnable AND FB_Schneider_EVLink_14.bEnableWrite;

FB_Schneider_EVLink_15.stSetupECS.byDisableSOC 	:= bySOC_D_CS_15;		   			
FB_Schneider_EVLink_15.stSetupECS.byEnableSOC 	:= bySOC_E_CS_15;	
FB_Schneider_EVLink_15.stSetupECS.byPriority 	:= byPrioCS_15;
FB_Schneider_EVLink_15.stSetupECS.rMaxPower 		:= rMaxPowerCS_15;
FB_Schneider_EVLink_15.stSetupECS.byCSMinPower	:= byMinPowerCS_15;
FB_Schneider_EVLink_15.bEnable					:= bEnabledCS_15;
FB_Schneider_EVLink_15.stSetupECS.bManualyOn		:= bChrgManuCS_15;
FB_Schneider_EVLink_15.stSetupECS.byManualyTargetPower := byChrgManuSPCS_15;

bIsEnabledCS_15 		:= FB_Schneider_EVLink_15.stDataECS.bEnabled;
byStateMinPowerCS_15 := FB_Schneider_EVLink_15.stDataECS.bySCSMinPower;
rTargetPowerCS_15 	:= FB_Schneider_EVLink_15.stDataECS.rTargetPower;	
byErrorWarningCS_15 	:= FB_Schneider_EVLink_15.stDataECS.byErrorWarning;
bCarConnectedCS_15 	:= FB_Schneider_EVLink_15.stDataECS.bCarConnected;
rChrgTimeCS_15 		:= FB_Schneider_EVLink_15.stDataECS.arrChargingTimeInMin[1];
lr_CSPower_15 		:= FB_Schneider_EVLink_15.stDataElectric.lrPowerTotal;
bStateOkCS_15		:= FB_Schneider_EVLink_15.bEnable AND FB_Schneider_EVLink_15.bEnableWrite;

FB_Schneider_EVLink_16.stSetupECS.byDisableSOC 	:= bySOC_D_CS_16;		   			
FB_Schneider_EVLink_16.stSetupECS.byEnableSOC 	:= bySOC_E_CS_16;	
FB_Schneider_EVLink_16.stSetupECS.byPriority 	:= byPrioCS_16;
FB_Schneider_EVLink_16.stSetupECS.rMaxPower 		:= rMaxPowerCS_16;
FB_Schneider_EVLink_16.stSetupECS.byCSMinPower	:= byMinPowerCS_16;
FB_Schneider_EVLink_16.bEnable					:= bEnabledCS_16;
FB_Schneider_EVLink_16.stSetupECS.bManualyOn		:= bChrgManuCS_16;
FB_Schneider_EVLink_16.stSetupECS.byManualyTargetPower := byChrgManuSPCS_16;

bIsEnabledCS_16 		:= FB_Schneider_EVLink_16.stDataECS.bEnabled;
byStateMinPowerCS_16 := FB_Schneider_EVLink_16.stDataECS.bySCSMinPower;
rTargetPowerCS_16 	:= FB_Schneider_EVLink_16.stDataECS.rTargetPower;	
byErrorWarningCS_16 	:= FB_Schneider_EVLink_16.stDataECS.byErrorWarning;
bCarConnectedCS_16 	:= FB_Schneider_EVLink_16.stDataECS.bCarConnected;
rChrgTimeCS_16 		:= FB_Schneider_EVLink_16.stDataECS.arrChargingTimeInMin[1];
lr_CSPower_16 		:= FB_Schneider_EVLink_16.stDataElectric.lrPowerTotal;
bStateOkCS_16		:= FB_Schneider_EVLink_16.bEnable AND FB_Schneider_EVLink_16.bEnableWrite;

FB_Schneider_EVLink_17.stSetupECS.byDisableSOC 	:= bySOC_D_CS_17;		   			
FB_Schneider_EVLink_17.stSetupECS.byEnableSOC 	:= bySOC_E_CS_17;	
FB_Schneider_EVLink_17.stSetupECS.byPriority 	:= byPrioCS_17;
FB_Schneider_EVLink_17.stSetupECS.rMaxPower 		:= rMaxPowerCS_17;
FB_Schneider_EVLink_17.stSetupECS.byCSMinPower	:= byMinPowerCS_17;
FB_Schneider_EVLink_17.bEnable					:= bEnabledCS_17;
FB_Schneider_EVLink_17.stSetupECS.bManualyOn		:= bChrgManuCS_17;
FB_Schneider_EVLink_17.stSetupECS.byManualyTargetPower := byChrgManuSPCS_17;

bIsEnabledCS_17 		:= FB_Schneider_EVLink_17.stDataECS.bEnabled;
byStateMinPowerCS_17 := FB_Schneider_EVLink_17.stDataECS.bySCSMinPower;
rTargetPowerCS_17 	:= FB_Schneider_EVLink_17.stDataECS.rTargetPower;	
byErrorWarningCS_17 	:= FB_Schneider_EVLink_17.stDataECS.byErrorWarning;
bCarConnectedCS_17 	:= FB_Schneider_EVLink_17.stDataECS.bCarConnected;
rChrgTimeCS_17 		:= FB_Schneider_EVLink_17.stDataECS.arrChargingTimeInMin[1];
lr_CSPower_17 		:= FB_Schneider_EVLink_17.stDataElectric.lrPowerTotal;
bStateOkCS_17		:= FB_Schneider_EVLink_17.bEnable AND FB_Schneider_EVLink_17.bEnableWrite;

FB_Schneider_EVLink_18.stSetupECS.byDisableSOC 	:= bySOC_D_CS_18;		   			
FB_Schneider_EVLink_18.stSetupECS.byEnableSOC 	:= bySOC_E_CS_18;	
FB_Schneider_EVLink_18.stSetupECS.byPriority 	:= byPrioCS_18;
FB_Schneider_EVLink_18.stSetupECS.rMaxPower 		:= rMaxPowerCS_18;
FB_Schneider_EVLink_18.stSetupECS.byCSMinPower	:= byMinPowerCS_18;
FB_Schneider_EVLink_18.bEnable					:= bEnabledCS_18;
FB_Schneider_EVLink_18.stSetupECS.bManualyOn		:= bChrgManuCS_18;
FB_Schneider_EVLink_18.stSetupECS.byManualyTargetPower := byChrgManuSPCS_18;

bIsEnabledCS_18 		:= FB_Schneider_EVLink_18.stDataECS.bEnabled;
byStateMinPowerCS_18 := FB_Schneider_EVLink_18.stDataECS.bySCSMinPower;
rTargetPowerCS_18 	:= FB_Schneider_EVLink_18.stDataECS.rTargetPower;	
byErrorWarningCS_18 	:= FB_Schneider_EVLink_18.stDataECS.byErrorWarning;
bCarConnectedCS_18 	:= FB_Schneider_EVLink_18.stDataECS.bCarConnected;
rChrgTimeCS_18 		:= FB_Schneider_EVLink_18.stDataECS.arrChargingTimeInMin[1];
lr_CSPower_18 		:= FB_Schneider_EVLink_18.stDataElectric.lrPowerTotal;
bStateOkCS_18		:= FB_Schneider_EVLink_18.bEnable AND FB_Schneider_EVLink_18.bEnableWrite;


// calculate House Power   (Gesamt Bezug + PV Produktion - EV Lesitung Summe)
r_House := GVL.ELEKTRO_1_Leistung + GVL.ELEKTRO_4_Leistung - LREAL_TO_REAL(lr_CSPowerTotal);

// send kWh counters to cloud

lr_EnergyCounterCS_1 := FB_Schneider_EVLink_1.fbCS.lrTotalCounterEnergy_Consumption;
lr_EnergyCounterCS_2 := FB_Schneider_EVLink_2.fbCS.lrTotalCounterEnergy_Consumption;
lr_EnergyCounterCS_3 := FB_Schneider_EVLink_3.fbCS.lrTotalCounterEnergy_Consumption;
lr_EnergyCounterCS_4 := FB_Schneider_EVLink_4.fbCS.lrTotalCounterEnergy_Consumption;
lr_EnergyCounterCS_5 := FB_Schneider_EVLink_5.fbCS.lrTotalCounterEnergy_Consumption;
lr_EnergyCounterCS_6 := FB_Schneider_EVLink_6.fbCS.lrTotalCounterEnergy_Consumption;
lr_EnergyCounterCS_7 := FB_Schneider_EVLink_7.fbCS.lrTotalCounterEnergy_Consumption;
lr_EnergyCounterCS_8 := FB_Schneider_EVLink_8.fbCS.lrTotalCounterEnergy_Consumption;
lr_EnergyCounterCS_9 := FB_Schneider_EVLink_9.fbCS.lrTotalCounterEnergy_Consumption;
lr_EnergyCounterCS_10 := FB_Schneider_EVLink_10.fbCS.lrTotalCounterEnergy_Consumption;
lr_EnergyCounterCS_11 := FB_Schneider_EVLink_11.fbCS.lrTotalCounterEnergy_Consumption;
lr_EnergyCounterCS_12 := FB_Schneider_EVLink_12.fbCS.lrTotalCounterEnergy_Consumption;
lr_EnergyCounterCS_13 := FB_Schneider_EVLink_13.fbCS.lrTotalCounterEnergy_Consumption;
lr_EnergyCounterCS_14 := FB_Schneider_EVLink_14.fbCS.lrTotalCounterEnergy_Consumption;
lr_EnergyCounterCS_15 := FB_Schneider_EVLink_15.fbCS.lrTotalCounterEnergy_Consumption;
lr_EnergyCounterCS_16 := FB_Schneider_EVLink_16.fbCS.lrTotalCounterEnergy_Consumption;
lr_EnergyCounterCS_17 := FB_Schneider_EVLink_17.fbCS.lrTotalCounterEnergy_Consumption;
lr_EnergyCounterCS_18 := FB_Schneider_EVLink_18.fbCS.lrTotalCounterEnergy_Consumption;

END_PROGRAM

// ---- Lynus/PrgEMS.TcPOU
PROGRAM PrgEMS
VAR PERSISTENT
	byMaxDepthOfDischrgEPO		: BYTE;							//{#lynus.ag#()}
	byPrioMinChrgBattSOCInEPO	: BYTE;							//{#lynus.ag#()}
	byResChrgfromGridToBatt		: BYTE;							//{#lynus.ag#()}
	byReserveSOCEPO				: BYTE;							//{#lynus.ag#()}
	uiUpdateTime				: UINT;							//{#lynus.ag#()}
	bEnableEMS					: BOOL;							//{#lynus.ag#()}
	bAllowChrgFromGrid			: BOOL;							//{#lynus.ag#()}
	rMainFuseCSEMS				: REAL;							//{#lynus.ag#()}
	iOperationModeEMS			: INT;							//{#lynus.ag#()}
	rSizeGridConn				: REAL;							//{#lynus.ag#()}
END_VAR
VAR
	fbEMS						: FB_EMS_V2;
	bIsEnableEMS				: BOOL;							//{#lynus.ag#()}
	bStateAllowChrgFromGrid		: BOOL;							//{#lynus.ag#()}
	bStateFuseCS				: BOOL;							//{#lynus.ag#()}
	bHPActivate					: BOOL;							//{#lynus.ag#()}
	bControllingState			: BOOL;							//{#lynus.ag#()}
	iMessageEMS					: INT;							//{#lynus.ag#()}
	rHeartbeatEMS				: REAL;							//{#lynus.ag#()}
	rErrorWarningEMS			: REAL;							//{#lynus.ag#()}
	rReadyEMS					: REAL;							//{#lynus.ag#()}
	rNewBatteryPowerEMS			: REAL;							//{#lynus.ag#()}
	fbGrid: FB_Grid_Power_Ext_Input;

END_VAR

IF iOperationModeEMS = 0 THEN fbEMS.eOperationMode := E_OperatingMode_EMS.eAllOff;
ELSIF iOperationModeEMS = 1 THEN fbEMS.eOperationMode := E_OperatingMode_EMS.eSelfConsumption;	
ELSIF iOperationModeEMS = 2 THEN fbEMS.eOperationMode := E_OperatingMode_EMS.ePeakLoadCapping;
ELSIF iOperationModeEMS = 3 THEN fbEMS.eOperationMode := E_OperatingMode_EMS.eLoadManagement;			
END_IF
fbEMS.stSetupEMS.bAllowChrgFromGrid := bAllowChrgFromGrid;
fbEMS.stSetupEMS.byMaxDepthOfDischrgEPO := byMaxDepthOfDischrgEPO;
// fbEMS.stSetupEMS.byPrioMinChrgBattSOCInEPO := byPrioMinChrgBattSOCInEPO;
// fbEMS.stSetupEMS.byResChrgfromGridToBatt := byResChrgfromGridToBatt;
fbEMS.stSetupEMS.byReserveSOCEPO := byReserveSOCEPO;
//fbEMS.stSetupEMS.rSizeMainFuseCS := rMainFuseCSEMS;
fbEMS.stSizeMainFuseCS.rElSizeLine1 := rMainFuseCSEMS;
fbEMS.stSetupEMS.bEnableMainFuseFunc := bStateFuseCS;
fbEMS.stSetupEMS.uiUpdateTime := uiUpdateTime;

fbEMS(
	bEnable						:= bEnableEMS, 
//	diNrOfEM_IN_ECS				:= , 
	stSetupEMS					:= , 
	eOperationMode				:= , 
	eSpeedModeBackendController	:= E_SpeedModeBackendController_EMS.eFast, 
	eSpeedModeLocalController	:= E_SpeedModeLocalController_EMS.eFast,
	bActivateHP					:= bHPActivate, 
	bControllingState			:= bControllingState, 
	rHeartbeat					:= rHeartbeatEMS, 
	rErrorWarning				:= rErrorWarningEMS, 
	rEnergyOptReady				:= rReadyEMS, 
	rNewBattPower				:= rNewBatteryPowerEMS, 

	eMessageEMS				=> iMessageEMS, 
	bStateEnable			=> bIsEnableEMS, 
	bStateAllowChrgFromGrid	=> bStateAllowChrgFromGrid, 
	bMissingPowerData		=> , 
	bSurplusAvailable		=> , 
	byProgress				=> , 
	uiState_OUT				=> , 
	diNrOfEMS_OUT			=> , 
	arrMinPrioReached		=> , 
	arrMaxPrioReached		=> ,
	);

								
fbGrid(
	bEnable:= TRUE, 
	diNrOfEMS_IN:= prgEMS.fbEMS.diNrOfEMS_OUT, 
	rSizeGridConn:= rSizeGridConn , 
	bExtErrorGrid:= , 
	lrExtGridPower:= GVL.ELEKTRO_1_Leistung , 
	lrExtTotalCounterEnergy_Consumption:= , 
	lrExtTotalCounterEnergy_Production:= , 
	lrExtCounterEnergyT1_Consumption:= , 
	lrExtCounterEnergyT2_Consumption:= , 
	lrExtCounterEnergyT1_Production:= , 
	lrExtCounterEnergyT2_Production:= , 
	stDataGrid=> , 
	diNrOfGrid_OUT=> );

END_PROGRAM
